TYPE McReadParameterArgs :
STRUCT
	///Number of the parameter
	parameterNumber: INT;
END_STRUCT
END_TYPE

(* stored: Version 1.1.0.1, ProductVersion 3.1.4019.2
   DUT McReadParameterArgs: Id {fc23405f-4e07-4fff-bd64-7e4ef31ed984} *)
